FUNCTION_BLOCK FB_ProtectRelay_DM2 EXTENDS FB_ProtectRelay_Base
//////////////////
// REF615 + REU615 : communication not allowed by EDF 

VAR_OUTPUT
	//Child objects

END_VAR

VAR_INPUT
	IN_AlarmIMax_IO								: BOOL; //Max I Alarm, Losing autorisation and not possible to consumed
	IN_AlarmUmin_IO									: BOOL; //Min U , Keeping autorisation, If we have 3 gte in 30 min ==> Stop fedding and consumed during 2h
	IN_MesWatchdogREU615_IO						: BOOL:=TRUE ;// Watchdog . 0= alarm
	MesDataExd		: ProtectRelay_Standard ; 	
END_VAR

VAR
	//M_ALARMMANAGEMENT VARIABLES//

	
	// EVALUATE //
	TON_GteIsLong	: TON ; 
	
	


		
END_VAR

METHOD M_AlarmManagement
//////////////////
// Manages Sepam Alarms. Alarms opens HT CB until Sepam manual Reset . Warning Opens CB-L but does not maintain warning
/////////////////

VAR 
	// Method local variables (reinitialized at each cycle) 
	FB_AlarmCodeManager 	: FB_AlarmCodeManager ; 

 
END_VAR


// ALARM CODE //
	FB_AlarmCodeManager(
		bAlarm1				:= MesDataExd.MesData.MesAlarmImax , 						// Max I>>0  fault 	 	
		bAlarm2				:= MesDataExd.MesData.MesAlarmUmin ,							// GTE fault 
		bAlarm3				:= MesDataExd.MesData.MesAlarmCom,						// Communication Alarm #COM
		bAlarm4				:= NOT IN_MesWatchDog_IO, 						// Watchdog REF615 not received      #COM 
		bAlarm5				:= NOT IN_MesWatchdogREU615_IO, 				// Watchdog REU615 not received	 #COM
		bAlarm6				:= FALSE, 									// 
		bAlarm7				:= FALSE, 									//
		bAlarm8				:= FALSE,                                   //
		bAlarm9				:= FALSE,                                   //
		bAlarm10			:= FALSE,                                   //
		bAlarm11			:= FALSE,                                   //
		bAlarm12			:= FALSE,                                   //
		bAlarm13			:= FALSE, 									//
		bAlarm14			:= FALSE, 									//
		bAlarm15			:= FALSE ,									// 
		wAlarmCode			=>MesDataExd.MesData.MesAlarmCode);

// WARNING CODE //
	FB_AlarmCodeManager(
		bAlarm1			:= FALSE , //
		bAlarm2			:= FALSE , //	
		bAlarm4			:= MesDataExd.MesData.MesAlarmUmin_Long, 						// GTE long 
		bAlarm5			:= FALSE, 									//
		bAlarm6			:= FALSE,                                   //
		bAlarm7			:= FALSE,                                   //
		bAlarm8			:= FALSE,                                   //
		bAlarm9			:= FALSE,                                   //
		bAlarm10		:= FALSE,                                   //
		bAlarm11		:= FALSE,                                   //
		bAlarm12		:= FALSE,                                   //
		bAlarm13		:= FALSE,                                   //
		bAlarm14		:= FALSE,                                   //
		bAlarm15		:= FALSE, 									//
		wAlarmCode		=>MesDataExd.MesData.MesWarningCode);

// EVENT CODE //
	FB_AlarmCodeManager(
		bAlarm1			:=FALSE, 		//  
		bAlarm2			:=FALSE, 		//  
		bAlarm3			:=FALSE, 		//  
		bAlarm4			:=FALSE, 		// 
		bAlarm5			:=FALSE,        //
		bAlarm6			:=FALSE,        //
		bAlarm7			:=FALSE,        //
		bAlarm8			:=FALSE,        //
		bAlarm9			:=FALSE,        //
		bAlarm10		:=FALSE,        //
		bAlarm11		:=FALSE,        //
		bAlarm12		:=FALSE,        //
		bAlarm13		:=FALSE,        //
		bAlarm14		:=FALSE,        //
		bAlarm15		:=FALSE, 
		wAlarmCode		=>MesDataExd.MesData.MesEventCode);
END_METHOD

METHOD M_CP
//////////////////
//  Emulator
/////////////////

VAR 
	// Method local variables (reinitialized at each cycle) 
	
END_VAR


SUPER^.M_CP() ; 




Trig_Cmd_Read(CLK:=IN_CmdToggleRead);
Trig_Cmd_Write(CLK:=IN_CmdToggleWrite);
	
IF Trig_Cmd_Read.Q THEN
	IN_CmdToggleRead := FALSE;
	MesDataExd.MesData.MesCP_Read := NOT MesDataExd.MesData.MesCP_Read;
END_IF


IF Trig_Cmd_Write.Q THEN
	IN_CmdToggleWrite := FALSE;
	MesDataExd.MesData.MesCP_Write := NOT MesDataExd.MesData.MesCP_Write;
END_IF
END_METHOD

METHOD M_Evaluate
VAR_INPUT
END_VAR
//Need to check the GTE FAULT


// GTE IS LONG AFTER 50S
TON_GteIsLong(IN:=IN_AlarmUmin_IO ,PT:=T#50S); 
MesDataExd.MesData.MesAlarmUmin_Long := TON_GteIsLong.Q ; 


//Update MesData

MesDataExd.MesData.MesAlarmUmin 			:= IN_AlarmUmin_IO;

TON_ComAlarm(IN:=NOT IN_MesWatchDog_IO OR NOT IN_MesWatchdogREU615_IO , PT:=ParamTempoComAlarm ) ; 
MesDataExd.MesData.MesAlarmCom		:=TON_ComAlarm.Q  ; 
MesDataExd.MesData.MesAlarmImax		:= IN_AlarmIMax_IO;
END_METHOD

END_FUNCTION_BLOCK

(* stored: Version 1.1.0.1, ProductVersion 3.1.4024.12
   POU FB_ProtectRelay_DM2: Id {9cf6550c-5f62-450e-8a26-31d4507a3632}, SpecialFunc None
   Method M_AlarmManagement: Id {28254a00-8506-4acf-a58d-02d5647dc1ec}
   Method M_CP: Id {65a19b94-7463-4c8b-bef2-181a419b7cfc}
   Method M_Evaluate: Id {9d2a05e2-f98c-4167-b791-289c9021cdda} *)
